Staubli VAL3: readFile.pgx

public program readFile(string x_sFilename, string& x_sLine[])
  local num l_nFileHandler
  local num l_nReadLines
  local num l_nDataSize
  local string l_sLine
begin

  // Open file to write
  l_nFileHandler = $fileOpen(x_sFilename, "r")
  // init Buffer sLine
  resize(x_sLine, 1, 1)
  x_sLine = ""
  l_nDataSize = 0
  // read line by line
  do
    l_nReadLines = $fileGet(l_nFileHandler,l_sLine,1)
    if l_nReadLines > 0
      append(x_sLine)
      x_sLine[l_nDataSize] = l_sLine
    endIf
    l_nDataSize = l_nDataSize + 1
  until l_nReadLines == 0

  // remove last entry in x_sLine, because of "append" command before
  resize(x_sLine, 1, size(x_sLine)-1)
  // close file
  $fileClose(l_nFileHandler)

end
